// Motor control interface — extends I_StateMachine
INTERFACE I_Motor EXTENDS I_StateMachine

METHOD Start : BOOL
VAR_INPUT
    fSpeed : LREAL; // Target speed [rpm]
END_VAR
END_METHOD

METHOD Stop : BOOL
VAR_INPUT
END_VAR
END_METHOD

METHOD GetSpeed : LREAL
VAR_INPUT
END_VAR
END_METHOD

METHOD IsRunning : BOOL
VAR_INPUT
END_VAR
END_METHOD

METHOD IsStopped : BOOL
VAR_INPUT
END_VAR
END_METHOD

END_INTERFACE

(* stored: Version 1.1.0.1, ProductVersion 3.1.4024.12
   Itf I_Motor: Id {45022258-330C-4C50-A85B-1B53BD811EF5}
   Method Start: Id {A1D8C5DC-9C7A-40CE-A31A-5DED4FB123D8}
   Method Stop: Id {7C5FA959-1E81-4DBF-AD15-58CB53596C4A}
   Method GetSpeed: Id {09CFA118-EAE7-4472-A985-E94AB2314797}
   Method IsRunning: Id {420633D5-4F5D-4750-A64E-08EB777AE159}
   Method IsStopped: Id {60E08564-7ABB-4903-A068-A8B16960DDEA} *)
